(* PLC project Sin nombre, Desconocido Sin nombre 1 *)
(* stored: creationDateTime 2023-09-25T11:39:21, modificationDateTime 2023-10-02T19:29:10 *)

PROGRAM program0
  VAR
    Sensor_Inc AT %IX0.3 : BOOL;
    Luz_verde AT %QX0.1 : BOOL;
    Luz_azul AT %QX0.2 : BOOL;
    Luz_roja AT %QX0.0 : BOOL;
  END_VAR
  VAR
    Retardo_LR : TIME := T#250ms;
    Retardo_LA : TIME := T#3s;
    TP0 : TP;
    TOF0 : TOF;
    TOF1 : TOF;
    CTU0 : CTU;
  END_VAR
  VAR  (* added by the conversion: wires and edge detectors of the diagram *)
    _NOT2_OUT : BOOL;
    _AND26_OUT : BOOL;
    R_TRIG1 : R_TRIG;
  END_VAR

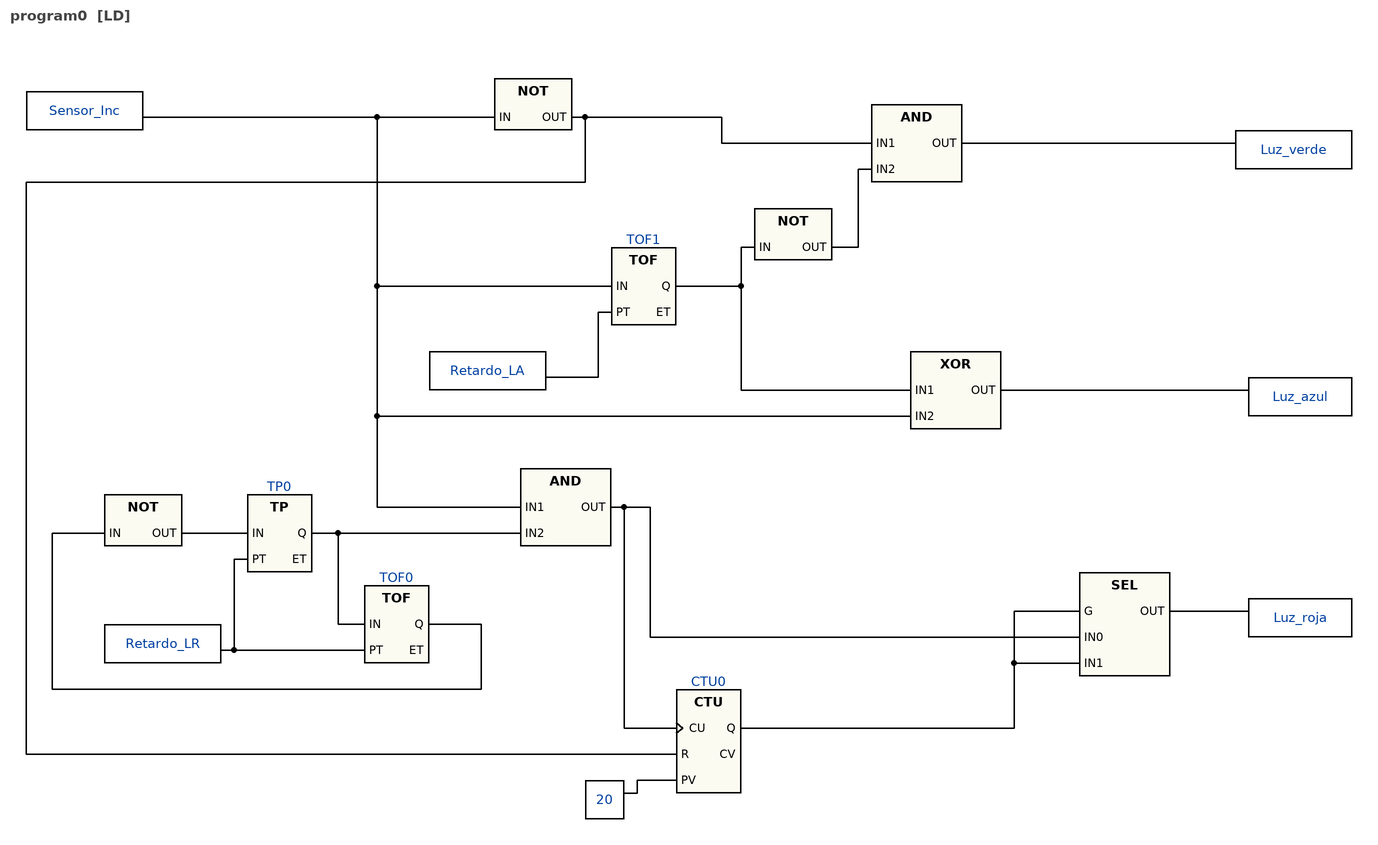
(* LD diagram, written out as Structured Text *)
_NOT2_OUT := NOT Sensor_Inc;
TOF1(IN := Sensor_Inc, PT := Retardo_LA);
Luz_verde := _NOT2_OUT AND NOT TOF1.Q;
Luz_azul := TOF1.Q XOR Sensor_Inc;
TOF0(IN := TP0.Q, PT := Retardo_LR);
TP0(IN := NOT TOF0.Q, PT := Retardo_LR);
_AND26_OUT := Sensor_Inc AND TP0.Q;
R_TRIG1(CLK := _AND26_OUT);
CTU0(CU := R_TRIG1.Q, R := _NOT2_OUT, PV := 20);
Luz_roja := SEL(CTU0.Q, _AND26_OUT, CTU0.Q);
END_PROGRAM

CONFIGURATION Config0
  RESOURCE Res0 ON PLC
    TASK task0(INTERVAL := T#20ms, PRIORITY := 0);
    PROGRAM instance0 WITH task0 : program0;
  END_RESOURCE
END_CONFIGURATION
